Omron CX-Programmer project NewProject (CX-Programmer 9.51)

# PLC my_first_project: CP1L L
; Comment

## Global symbols (name address type ; comment)
T0001 BOOL  ; Timer number

## Program NewProgram1 (cyclic task 0)
Local symbols
button_2 0.01 BOOL  ; comment
button_3 0.02 BOOL
out_2 100.01 BOOL

### Section Section1

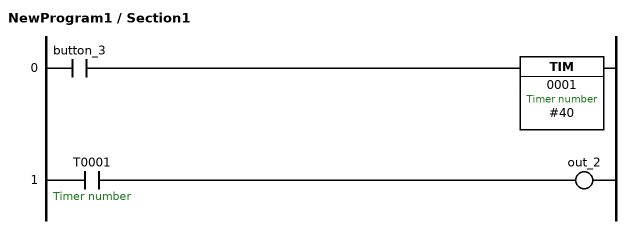
; rung 0
LD button_3
TIM 0001 #40  ; Timer number
; rung 1
LD T0001  ; Timer number
OUT out_2

### Section END
; rung 0
END(001)